FUNCTION_BLOCK FB_Sorter
VAR_INPUT
END_VAR
VAR_OUTPUT
END_VAR
VAR
	rTrigAtExit : Tc2_Standard.R_TRIG;
	atExitEdgeDetected : BOOL;
	
	
	Step_0: BOOL;
	Step_1 : BOOL;
	Step_2 : BOOL;
	Step_3 : BOOL;
	Step_4 : BOOL;
	Step_5 : BOOL;
	Step_6 : BOOL;
END_VAR
VAR_IN_OUT
	control_data : Plant_CTRL;
	control_data_vision : CM_Vision_UDT;
	control_data_Conveyor2 : CM_DO_UDT;
	
	control_data_sorter1 : CM_DO_UDT;
	control_data_sorter2 : CM_DO_UDT;
	control_data_sorter3 : CM_DO_UDT;
	
	control_data_atExit : CM_DIN_UDT;
	
	
END_VAR
VAR // added by the converter: edge detectors and wires of the graphical bodies
    _w1, _w2, _w3, _w4, _w5, _w6 : BOOL;
END_VAR

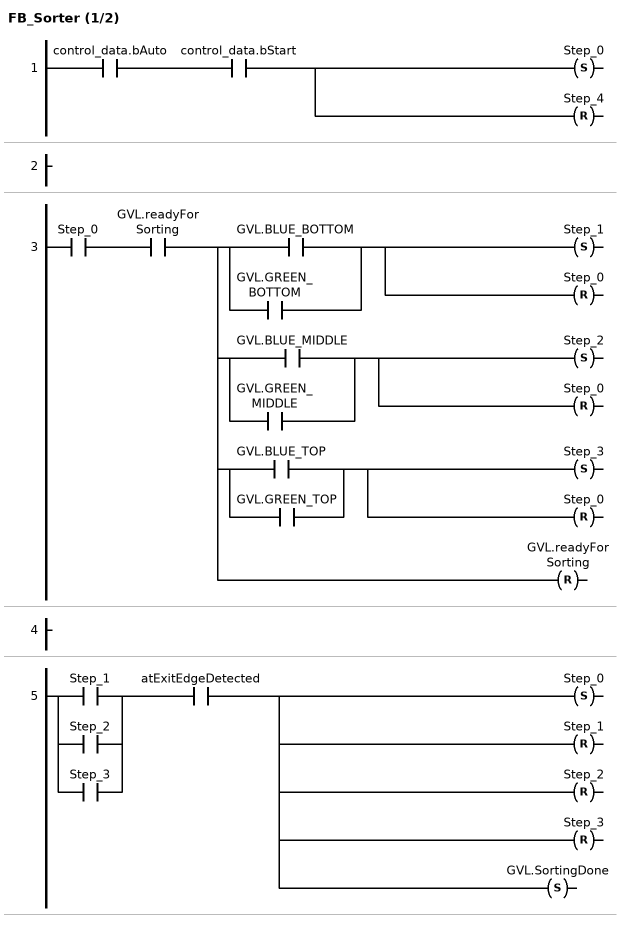
// NETWORK 1
_w1 := control_data.bAuto AND control_data.bStart;
Step_0 S= _w1;
Step_4 R= _w1;

// NETWORK 2

// NETWORK 3
_w2 := Step_0 AND GVL.readyForSorting;
_w3 := _w2 AND (GVL.BLUE_BOTTOM OR GVL.GREEN_BOTTOM);
Step_1 S= _w3;
Step_0 R= _w3;
_w4 := _w2 AND (GVL.BLUE_MIDDLE OR GVL.GREEN_MIDDLE);
Step_2 S= _w4;
Step_0 R= _w4;
_w5 := _w2 AND (GVL.BLUE_TOP OR GVL.GREEN_TOP);
Step_3 S= _w5;
Step_0 R= _w5;
GVL.readyForSorting R= _w2;

// NETWORK 4

// NETWORK 5
_w6 := (Step_1 OR Step_2 OR Step_3) AND atExitEdgeDetected;
Step_0 S= _w6;
Step_1 R= _w6;
Step_2 R= _w6;
Step_3 R= _w6;
GVL.SortingDone S= _w6;

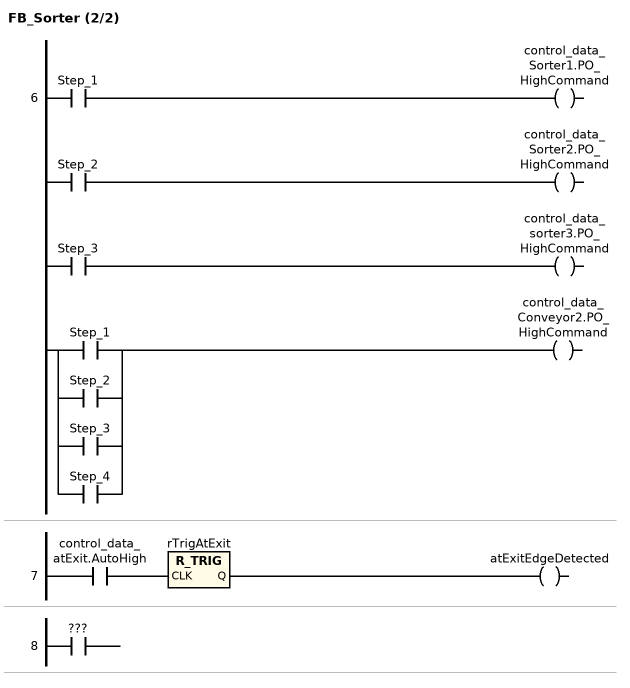
// NETWORK 6
control_data_Sorter1.PO_HighCommand := Step_1;
control_data_Sorter2.PO_HighCommand := Step_2;
control_data_sorter3.PO_HighCommand := Step_3;
control_data_Conveyor2.PO_HighCommand := Step_1 OR Step_2 OR Step_3 OR Step_4;

// NETWORK 7
rTrigAtExit(CLK := control_data_atExit.AutoHigh); // R_TRIG
atExitEdgeDetected := rTrigAtExit.Q;

// NETWORK 8

END_FUNCTION_BLOCK

(* stored: Version 1.1.0.1, ProductVersion 3.1.4024.13
   POU FB_Sorter: Id {495ed67c-a59d-48ee-aabf-bc1a273d4fac}, SpecialFunc None *)
